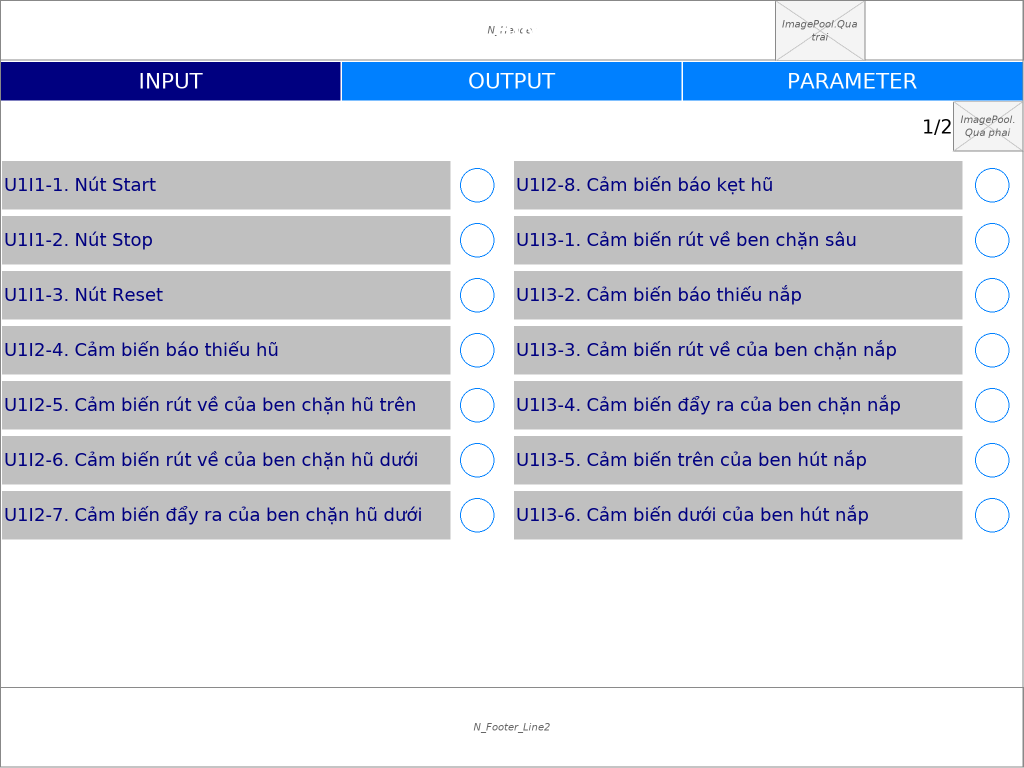
VISUALIZATION N_PLC_I2  // 1024x768
    Rectangle (886,102 103x50), "1/2"
    Frame (0,687 1024x80)
        shows N_Footer_Line2()
    Frame (0,0 1024x60)
        shows N_Header()
    Textfield (353,5 400x50), "MÀN HÌNH IO LINE 2"
    Image (775,0 90x61), image: ImagePool.Qua trai
        OnMouseClick: change screen: N_PLC_I1
    Rectangle (1,325 450x50), "U1I2-4. Cảm biến báo thiếu hũ"
    Rectangle (1,380 450x50), "U1I2-5. Cảm biến rút về của ben chặn hũ trên"
    Rectangle (1,435 450x50), "U1I2-6. Cảm biến rút về của ben chặn hũ dưới"
    Rectangle (1,490 450x50), "U1I2-7. Cảm biến đẩy ra của ben chặn hũ dưới"
    Rectangle (1,160 450x50), "U1I1-1. Nút Start"
    Rectangle (1,215 450x50), "U1I1-2. Nút Stop"
    Rectangle (1,270 450x50), "U1I1-3. Nút Reset"
    Ellipse (460,168 34x34), colour toggle: GVL_IO.bStart, input disabled if: true
    Ellipse (460,223 34x34), colour toggle: GVL_IO.bStop, input disabled if: true
    Ellipse (460,278 34x34), colour toggle: GVL_IO.bReset, input disabled if: true
    Ellipse (460,333 34x34), colour toggle: PR_Line02.fb_CupSupply.bCupEmpty, input disabled if: true
    Ellipse (460,388 34x34), colour toggle: PR_Line02.fb_CupSupply.fbCylinder_Up.bAtRetract, input disabled if: true
    Ellipse (460,443 34x34), colour toggle: PR_Line02.fb_CupSupply.fbCylinder_Dw.bAtRetract, input disabled if: true
    Ellipse (460,498 34x34), colour toggle: PR_Line02.fb_CupSupply.fbCylinder_Dw.bAtExtend, input disabled if: true
    Rectangle (513,490 450x50), "U1I3-6. Cảm biến dưới của ben hút nắp"
    Rectangle (513,160 450x50), "U1I2-8. Cảm biến báo kẹt hũ"
    Rectangle (513,215 450x50), "U1I3-1. Cảm biến rút về ben chặn sâu"
    Rectangle (513,270 450x50), "U1I3-2. Cảm biến báo thiếu nắp"
    Rectangle (513,325 450x50), "U1I3-3. Cảm biến rút về của ben chặn nắp"
    Rectangle (513,380 450x50), "U1I3-4. Cảm biến đẩy ra của ben chặn nắp"
    Rectangle (513,435 450x50), "U1I3-5. Cảm biến trên của ben hút nắp"
    Ellipse (975,168 34x34), colour toggle: PR_Line02.fb_CupSupply.bCupDrop, input disabled if: true
    Ellipse (975,498 34x34), colour toggle: PR_Line02.fb_LidSupply.fbCylinder_Suction.bAtExtend, input disabled if: true
    Ellipse (975,223 34x34), colour toggle: PR_Line02.fb_WormWeight.fbCylinder.bAtRetract, input disabled if: true
    Ellipse (975,278 34x34), colour toggle: PR_Line02.fb_LidSupply.bLidEmpty, input disabled if: true
    Ellipse (975,333 34x34), colour toggle: PR_Line02.fb_LidSupply.fbCylinder_LidStopper.bAtRetract, input disabled if: true
    Ellipse (975,388 34x34), colour toggle: PR_Line02.fb_LidSupply.fbCylinder_LidStopper.bAtExtend, input disabled if: true
    Ellipse (975,443 34x34), colour toggle: PR_Line02.fb_LidSupply.fbCylinder_Suction.bAtRetract, input disabled if: true
    Image (953,101 70x50), image: ImagePool.Qua phai
        OnMouseClick: change screen: N_PLC_I2_next
    Rectangle (0,61 341x40), "INPUT"
        OnMouseClick: change screen: N_PLC_I2
    Rectangle (341,61 341x40), "OUTPUT"
        OnMouseClick: change screen: N_PLC_O2
    Rectangle (682,61 341x40), "PARAMETER"
        OnMouseClick: change screen: N_Parameter_2
END_VISUALIZATION

(* stored: Version 1.1.0.1, ProductVersion 3.1.4024.12
   Visu N_PLC_I2: Id {e46e315c-264f-43f7-ba82-8efd9c9a7853} *)
